// TIA Portal V20 export
TYPE "LER_typeHipotTrackingData"
// stored: Access Published
   STRUCT
      resultDataOhm { ExternalWritable := 'False'} : String[5];
      resultDataCapa { ExternalWritable := 'False'} : String[10];
      resultDataBddCount { ExternalWritable := 'False'} : String;
      resultDataBDD { ExternalWritable := 'False'} : "LER_typeHipotBddData";
      resultOK { ExternalWritable := 'False'} : Bool;
      resultNG { ExternalWritable := 'False'} : Bool;
      complete { ExternalWritable := 'False'} : Bool;
   END_STRUCT;
END_TYPE
